// TIA Portal V20 export
VAR_GLOBAL   // PLC tag table "Default tag table"
   SynchronousAxis_Slave_cam_Actor_Interface_AddressIn AT %I336.0 : "PD_TEL105_IN";
   PositioningAxis_Actor_Interface_AddressIn AT %I286.0 : "PD_TEL105_IN";
   SynchronousAxis_1_Actor_Interface_AddressIn AT %I330.0 : "PD_TEL105_IN";
   SynchronousAxis_2_Actor_Interface_AddressIn AT %I280.0 : "PD_TEL105_IN";
   SynchronousAxis_Slave_cam_Actor_Interface_AddressOut AT %Q266.0 : "PD_TEL105_OUT";
   PositioningAxis_Actor_Interface_AddressOut AT %Q286.0 : "PD_TEL105_OUT";
   SynchronousAxis_1_Actor_Interface_AddressOut AT %Q260.0 : "PD_TEL105_OUT";
   SynchronousAxis_2_Actor_Interface_AddressOut AT %Q280.0 : "PD_TEL105_OUT";
   "SynchronousAxis_2_Actor_Interface_AddressOut(1)" AT %Q330.0 : "PD_TEL105_OUT";
   "SynchronousAxis_1_Actor_Interface_AddressIn(1)" AT %I300.0 : "PD_TEL105_IN";
   "SynchronousAxis_1_Actor_Interface_AddressOut(1)" AT %Q300.0 : "PD_TEL105_OUT";
   STSRT_ AT %M1.0 : Bool;
END_VAR
